FUNCTION (*FUNCTION_NAME*) : TOD
VAR_INPUT
   day   : USINT;
   month : USINT;
END_VAR
VAR
(*VAR*)
END_VAR


IF (day   > 31) OR (day   = 0) THEN day   := 1; END_IF
IF (month > 12) OR (month = 0) THEN month := 1; END_IF


(*FUNCTION_NAME*) := (*VARNAME*)[month][day];

END_FUNCTION

(* stored: Version 1.1.0.1
   POU ( *FUNCTION_NAME* ): SpecialFunc None *)
